// TwinCAT 3 PLC project Beispielprojekt
// ProgramVersion: 3.1.4023.0
// libraries:
//   Lynus Energy Basic, * (Lynus AG)
//   Lynus Energy ModbusTCP, * (Lynus AG)
//   Lynus Persistent Data V1, * (Lynus AG)
//   Lynus Standards, * (Lynus AG)
//   Tc2_Standard, * (Beckhoff Automation GmbH)
//   Tc2_System, * (Beckhoff Automation GmbH)
//   Tc3_Module, * (Beckhoff Automation GmbH)
//   TSG Communicator, * (EfficientIO)
// project tree:
//   / FastTask.TcTTO, PlcTask.TcTTO, SlowTask.TcTTO
//   POUs/ prgCom.TcPOU, prgCS1.TcPOU, prgEM.TcPOU, prgEMS.TcPOU (not stored), prgGrid.TcPOU, prgPD.TcPOU, prgPV.TcPOU, prgVar.TcPOU
// real-time tasks:
//   TASK FastTask: cycle T#5ms, priority 4, ADS port 350
//   TASK PlcTask: cycle T#10ms, priority 8, ADS port 351
//   TASK SlowTask: cycle T#20ms, priority 12, ADS port 352
//   TASK PlcTask1: cycle T#10ms, priority 10, ADS port 353

CONFIGURATION Beispielprojekt
    RESOURCE PLC ON TwinCAT3
        TASK FastTask(INTERVAL := T#5ms, PRIORITY := 4);
        TASK PlcTask(INTERVAL := T#10ms, PRIORITY := 8);
        TASK SlowTask(INTERVAL := T#20ms, PRIORITY := 12);
        PROGRAM prgVar WITH FastTask : prgVar;
        PROGRAM prgCS1 WITH PlcTask : prgCS1;
        PROGRAM prgEMS WITH PlcTask : prgEMS;
        PROGRAM prgGrid WITH PlcTask : prgGrid;
        PROGRAM prgPD WITH PlcTask : prgPD;
        PROGRAM prgPV WITH PlcTask : prgPV;
        PROGRAM prgEM WITH PlcTask : prgEM;
        PROGRAM prgCom WITH SlowTask : prgCom;
    END_RESOURCE
END_CONFIGURATION

// ---- POUs/prgVar.TcPOU
PROGRAM prgVar
VAR
	fbVar			: FB_VarInfo;
	fbrw1			: FB_ReadWrite;
END_VAR

fbVar(
	bReadInfo:= , 
	eTMCFile:= eSelectTMCFile.eUseTMCFile, 
	eSavePositionTMCFile:= eSavePositionOnPLC.ePostionC, 
	udiCounterFoundVariables=> , 
	bError=> , 
	bBusy=> , 
	byProgress=> , 
	udiErrorCodeOut=> , 
	eErrorVarInfo_Out=> , 
	sVarWithError=> );
	
fbrw1();

END_PROGRAM

// ---- POUs/prgCS1.TcPOU
PROGRAM prgCS1
VAR
	fbApliT_1						: FB_ECS_Alpitronic_Hypercharger;
		
	bSManualyOn_DC_1				: BOOL;												//{#lynus.ag#()}
	bEnabled_DC_1					: BOOL;												//{#lynus.ag#()}
	bySManualyTargetPowerDC_1		: BYTE;												//{#lynus.ag#()}
	bySMinPowerECSDC_1				: BYTE;												//{#lynus.ag#()}
	byErrorWarningDC_1				: BYTE;												//{#lynus.ag#()}
	lrPowerTotalDC1					: LREAL;											//{#lynus.ag#()}
	lrPowerDC1_S1					: LREAL;											//{#lynus.ag#()}
	lrPowerDC1_S2					: LREAL;											//{#lynus.ag#()}
	rChargingTimeInMinDC1_S1		: REAL;												//{#lynus.ag#()}
	rChargingTimeInMinDC1_S2		: REAL;												//{#lynus.ag#()}
	rTargetPowerDC1					: REAL;												//{#lynus.ag#()}
	dwSOCCarDC1_S1					: DWORD;											//{#lynus.ag#()}
	dwSOCCarDC1_S2					: DWORD;											//{#lynus.ag#()}
	wStateDC1_S1					: WORD;												//{#lynus.ag#()}
	wStateDC1_S2					: WORD;												//{#lynus.ag#()}
	lrEnergySessionDC1_S1			: LREAL;											//{#lynus.ag#()}
	lrEnergySessionDC1_S2			: LREAL;											//{#lynus.ag#()}
	lrTotalEnergyDC1				: LREAL;											//{#lynus.ag#()}

	fbAlfen_1						: FB_ECS_Alfen_NG9xx_Platform;
		
	bSManualyOn_Alfen_1				: BOOL;												//{#lynus.ag#()}
	bEnabled_Alfen_1				: BOOL;												//{#lynus.ag#()}
	bySManualyTargetPower_Alfen_1	: BYTE;												//{#lynus.ag#()}
	bySMinPowerECS_Alfen_1			: BYTE;												//{#lynus.ag#()}
	byErrorWarning_Alfen_1			: BYTE;												//{#lynus.ag#()}
	lrPowerTotal_Alfen_1			: LREAL;											//{#lynus.ag#()}
	lrPower_Alfen_1_S1				: LREAL;											//{#lynus.ag#()}
	lrPower_Alfen_1_S2				: LREAL;											//{#lynus.ag#()}
	rChargingTimeInMin_Alfen_1_S1	: REAL;												//{#lynus.ag#()}
	rChargingTimeInMin_Alfen_1_S2	: REAL;												//{#lynus.ag#()}
	rTargetPower_Alfen_1			: REAL;												//{#lynus.ag#()}
	wState_Alfen_1_S1				: WORD;												//{#lynus.ag#()}
	wState_Alfen_1_S2				: WORD;												//{#lynus.ag#()}
	lrEnergySession_Alfen_1_S1		: LREAL;											//{#lynus.ag#()}
	lrEnergySession_Alfen_1_S2		: LREAL;											//{#lynus.ag#()}
	lrTotalEnergy_Alfen_1			: LREAL;											//{#lynus.ag#()}
	diff_netz_pv					: LREAL;											//{#lynus.ag#()}
END_VAR
VAR PERSISTENT
	bEnableDC1						: BOOL;												//{#lynus.ag#()}
	bManualyOnDC_1					: BOOL;												//{#lynus.ag#()}
	byMinPowerDC1					: BYTE;												//{#lynus.ag#()}
	byManualyTargetPowerDC_1		: BYTE;												//{#lynus.ag#()}
	byPrioDC1						: BYTE;												//{#lynus.ag#()}
	bySOCEnableDC1					: BYTE;												//{#lynus.ag#()}
	bySOCDisableDC1					: BYTE;												//{#lynus.ag#()}
	rMaxPowerDC1					: REAL;												//{#lynus.ag#()}
	
	bEnable_Alfen_1					: BOOL;												//{#lynus.ag#()}
	bManualyOn_Alfen_1				: BOOL;												//{#lynus.ag#()}
	byMinPower_Alfen_1				: BYTE;												//{#lynus.ag#()}
	byManualyTargetPower_Alfen_1	: BYTE;												//{#lynus.ag#()}
	byPrio_Alfen_1					: BYTE;												//{#lynus.ag#()}
	bySOCEnable_Alfen_1				: BYTE;												//{#lynus.ag#()}
	bySOCDisable_Alfen_1			: BYTE;												//{#lynus.ag#()}
	rMaxPower_Alfen_1				: REAL;												//{#lynus.ag#()}
END_VAR

(*-----------------------------------------------------------------------PV vs. Netzbezug------------------------------------------------------*)
IF (lrPowerTotalDC1 + lrPowerTotal_Alfen_1) > 0 AND prgPV.lrPowerPV > (lrPowerTotalDC1 + lrPowerTotal_Alfen_1) THEN diff_netz_pv := (lrPowerTotalDC1 + lrPowerTotal_Alfen_1);
ELSIF (lrPowerTotalDC1 + lrPowerTotal_Alfen_1) > 0 AND prgPV.lrPowerPV < (lrPowerTotalDC1 + lrPowerTotal_Alfen_1) THEN diff_netz_pv := prgPV.lrPowerPV;
ELSE diff_netz_pv := 0;
END_IF

(*-----------------------------------------------------------------------Alpitronic------------------------------------------------------*)
//Manual Power
fbApliT_1.stSetupECS.bManualyOn := bManualyOnDC_1;
	fbApliT_1.stSetupECS.byManualyTargetPower := byManualyTargetPowerDC_1;
		fbApliT_1.stSetupECS.byPriority := byPrioDC1;
			fbApliT_1.stSetupECS.byEnableSOC := bySOCEnableDC1;
				fbApliT_1.stSetupECS.byDisableSOC := bySOCDisableDC1;
					fbApliT_1.stSetupECS.rMaxPower := rMaxPowerDC1;
						fbApliT_1.stSetupECS.byCSMinPower := byMinPowerDC1;	
	
fbApliT_1(
	bEnable:= bEnableDC1, 
	bPowerDataInvers:= , 
	byElectricFuseLine:= , 
	byUnitID:= 1, 	//Normaly always 1 for Alpitronic
	diNrOfEMS_IN:= prgEMS.fbEMS.diNrOfEMS_OUT, 
	diNrOfEM_IN_CS:= , 
	sIPAdress:= '172.16.1.110', 
	stSetupECS:= , 
	stDataECS=> , 
	diNrOfECS_OUT=> );

bSManualyOn_DC_1 := fbApliT_1.stDataECS.bSManualyOn;
	bySManualyTargetPowerDC_1 := fbApliT_1.stDataECS.bySManualyTargetPower;
		byErrorWarningDC_1 := fbApliT_1.stDataECS.byErrorWarning;
			lrPowerTotalDC1 := fbApliT_1.stDataECS.lrTotalPower;
				lrPowerDC1_S1 :=  fbApliT_1.stDataECS.arrSocketPower[1];
					lrPowerDC1_S2 :=  fbApliT_1.stDataECS.arrSocketPower[2];	 	
						rChargingTimeInMinDC1_S1 := fbApliT_1.stDataECS.arrChargingTimeInMin[1];	
							rChargingTimeInMinDC1_S2 := fbApliT_1.stDataECS.arrChargingTimeInMin[2];
								dwSOCCarDC1_S1 := fbApliT_1.stDataECS.arrSocketSOCCar[1]; 
									dwSOCCarDC1_S2 := fbApliT_1.stDataECS.arrSocketSOCCar[2]; 	
										wStateDC1_S1 := fbApliT_1.stDataECS.arrSocketStateECS[1];
											wStateDC1_S2 := fbApliT_1.stDataECS.arrSocketStateECS[2];
												lrEnergySessionDC1_S1 := fbApliT_1.stDataECS.arrSocketEnergySession[1];
													lrEnergySessionDC1_S2 := fbApliT_1.stDataECS.arrSocketEnergySession[2];
														lrTotalEnergyDC1 := fbApliT_1.stDataECS.lrTotalCounterEnergy_Consumption;
															bySMinPowerECSDC_1 := fbApliT_1.stDataECS.bySCSMinPower;
																rTargetPowerDC1 := fbApliT_1.stDataECS.rTargetPower;
																	bEnabled_DC_1 := fbApliT_1.stDataECS.bEnabled;
																	
(*-----------------------------------------------------------------------Alfen------------------------------------------------------*)

//Manual Power
fbAlfen_1.stSetupECS.bManualyOn := bManualyOn_Alfen_1;
	fbAlfen_1.stSetupECS.byManualyTargetPower := byManualyTargetPower_Alfen_1;
		fbAlfen_1.stSetupECS.byPriority := byPrio_Alfen_1;
			fbAlfen_1.stSetupECS.byEnableSOC := bySOCEnable_Alfen_1;
				fbAlfen_1.stSetupECS.byDisableSOC := bySOCDisable_Alfen_1;
					fbAlfen_1.stSetupECS.rMaxPower := rMaxPower_Alfen_1;
						fbAlfen_1.stSetupECS.byCSMinPower := byMinPower_Alfen_1;	
	
fbAlfen_1(
	bEnable:= bEnable_Alfen_1, 
	bPowerDataInvers:= , 
	byElectricFuseLine:= , 
	byUnitID_Socket1:= 1, 
	byUnitID_Socket2:= 2, 
	byNumberOfSockets:= 2,		//1 or 2. Depends on whether it is a single or double charging station  
	byNumberOfConnectionWire:= 2, //1 or 2.  Depends on whether the charging station is supplied via a supply line or
	diNrOfEMS_IN:= prgEMS.fbEMS.diNrOfEMS_OUT, 
	diNrOfEM_IN_CS:= , 
	sIPAdress:= '172.16.1.100', 
	stSetupECS:= , 
	stDataECS=> , 
	diNrOfECS_OUT=> , 
	lrTotalPowerECSRealTime=> );						
						
bSManualyOn_Alfen_1 := fbAlfen_1.stDataECS.bSManualyOn;
	bySManualyTargetPower_Alfen_1 := fbAlfen_1.stDataECS.bySManualyTargetPower;
		byErrorWarning_Alfen_1 := fbAlfen_1.stDataECS.byErrorWarning;
			lrPowerTotal_Alfen_1 := fbAlfen_1.stDataECS.lrTotalPower;
				lrPower_Alfen_1_S1 :=  fbAlfen_1.stDataECS.arrSocketPower[1];
				lrPower_Alfen_1_S2 :=  fbAlfen_1.stDataECS.arrSocketPower[2];
					rChargingTimeInMin_Alfen_1_S1 := fbAlfen_1.stDataECS.arrChargingTimeInMin[1];
					rChargingTimeInMin_Alfen_1_S2 := fbAlfen_1.stDataECS.arrChargingTimeInMin[2];	
						wState_Alfen_1_S1 := fbAlfen_1.stDataECS.arrSocketStateECS[1];
						wState_Alfen_1_S2 := fbAlfen_1.stDataECS.arrSocketStateECS[2];
							lrEnergySession_Alfen_1_S1 := fbAlfen_1.stDataECS.arrSocketEnergySession[1];
							lrEnergySession_Alfen_1_S1 := fbAlfen_1.stDataECS.arrSocketEnergySession[2];
								lrTotalEnergy_Alfen_1 := fbAlfen_1.stDataECS.lrTotalCounterEnergy_Consumption;
									bySMinPowerECS_Alfen_1 := fbAlfen_1.stDataECS.bySCSMinPower;
										rTargetPower_Alfen_1 := fbAlfen_1.stDataECS.rTargetPower;
											bEnabled_Alfen_1 := fbAlfen_1.stDataECS.bEnabled;

END_PROGRAM

// ---- POUs/prgPV.TcPOU
PROGRAM prgPV
VAR
	fbPV1					: FB_Firmer_PV_Inverter_Sunspec;
	fbPV2					: FB_Firmer_PV_Inverter_Sunspec;
	fbPVInt1				: FB_PV_Power;
	fbPVInt2				: FB_PV_Power;
	fbPVCounter				: FB_EnergyCounter;
	lrPowerPV				: LREAL;				//{#lynus.ag#()}
	lrPowerPV1				: LREAL;				//{#lynus.ag#()}
	lrPowerPV2				: LREAL;				//{#lynus.ag#()}
	byErrorWarningPV1		: BYTE;					//{#lynus.ag#()}
	byErrorWarningPV2		: BYTE;					//{#lynus.ag#()}
END_VAR
VAR PERSISTENT
	lrCounterPV				: LREAL;				//{#lynus.ag#()}
END_VAR

fbPV1(
	bEnable:= TRUE, 
	sIPAdress:= '172.16.1.161',
	byUnitID_Inverter := 1,
	stFirmerInverterData=> , 
	stDataEMPower_PV=> , 
	stDataEMCounter_PV=> , 
	diNrOfEM_OUT_PV=> );

fbPV2(
	bEnable:= TRUE, 
	sIPAdress:= '172.16.1.162',
	byUnitID_Inverter := 1,
	stFirmerInverterData=> , 
	stDataEMPower_PV=> , 
	stDataEMCounter_PV=> , 
	diNrOfEM_OUT_PV=> );
	
fbPVInt1(
	bEnable:= TRUE, 
	bPowerDataInvers:= , 
	diNrOfEM_IN_PV:= fbPV1.diNrOfEM_OUT_PV, 
	stDataPv=> , 
	diNrOfPv_OUT=> );

fbPVInt2(
	bEnable:= TRUE, 
	bPowerDataInvers:= , 
	diNrOfEM_IN_PV:= fbPV2.diNrOfEM_OUT_PV, 
	stDataPv=> , 
	diNrOfPv_OUT=> );

lrPowerPV1 := fbPVInt1.stDataPv.lrPower;
lrPowerPV2 := fbPVInt2.stDataPv.lrPower;
	byErrorWarningPV1 := fbPVInt1.stDataPv.byErrorWarning;
	byErrorWarningPV2 := fbPVInt2.stDataPv.byErrorWarning;

// PV Power Total
lrPowerPV := fbPVInt1.stDataPv.lrPower + fbPVInt2.stDataPv.lrPower;


// EnergyCounter (Total)
fbPVCounter(
	byActiveTariff:= 1, 
	lrPowerInput:= 0 - lrPowerPV, 
	lrTotalCounterEnergy_Consumption=> , 
	lrTotalCounterEnergy_Production=> , 
	lrCounterEnergyT1_Consumption=> , 
	lrCounterEnergyT2_Consumption=> , 
	lrCounterEnergyT1_Production=> , 
	lrCounterEnergyT2_Production=> );
	
IF fbPVCounter.lrTotalCounterEnergy_Production > lrCounterPV THEN  	
	lrCounterPV := fbPVCounter.lrTotalCounterEnergy_Production;
END_IF

END_PROGRAM

// ---- POUs/prgGrid.TcPOU
PROGRAM prgGrid
VAR PERSISTENT
	rSizeGridConn				: REAL;									//{#lynus.ag#()}
END_VAR
VAR
	fbGrid						: FB_Grid_Power_Ext_Input;
	lrGridPower					: LREAL;								//{#lynus.ag#()}
END_VAR

IF prgEM.fbEM.stDataEMPowerRealTime.byErrorWarning = 2 THEN fbGrid.bExtErrorGrid := TRUE; ELSE fbGrid.bExtErrorGrid := FALSE; END_IF

fbGrid(
	bEnable:= TRUE, 
	diNrOfEMS_IN:= prgEMS.fbEMS.diNrOfEMS_OUT, 
	rSizeGridConn:= rSizeGridConn, 
	bExtErrorGrid:= , 
	lrExtGridPower:= prgEM.fbEM.stDataEMPowerRealTime.lrPowerTotal, 
	lrExtTotalCounterEnergy_Consumption:= 0, 
	lrExtTotalCounterEnergy_Production:= 0, 
	lrExtCounterEnergyT1_Consumption:= 0, 
	lrExtCounterEnergyT2_Consumption:= 0, 
	lrExtCounterEnergyT1_Production:= 0, 
	lrExtCounterEnergyT2_Production:= 0,
	stDataGrid=> ,
	diNrOfGrid_OUT=> );
	
lrGridPower := fbGrid.stDataGrid.lrPower;

END_PROGRAM

// ---- POUs/prgEM.TcPOU
PROGRAM prgEM
VAR
	fbEM				: FB_PhoenixContact_EM_EEM_EM375;
	lrEMPowerTotal		: LREAL;
END_VAR
VAR PERSISTENT
	bEnableEM			: BOOL;
	lrEMCounterProd		: LREAL;
	lrEMCounterCons		: LREAL;
END_VAR

fbEM(
	bEnable:=bEnableEM,
	byUnitID:=255,
	sIPAdress:='172.16.1.151',
	diNrOfEM_OUT=>,
	stDataEMPowerRealTime=>,
	stDataEMCounterRealTime=>);

lrEMPowerTotal := fbEM.stDataEMPowerRealTime.lrPowerTotal;
	lrEMCounterProd := fbEM.stDataEMCounterRealTime.lrTotalCounterEnergy_Production;
		lrEMCounterCons := fbEM.stDataEMCounterRealTime.lrTotalCounterEnergy_Consumption;

END_PROGRAM

// ---- POUs/prgPD.TcPOU
PROGRAM prgPD
VAR
	fbPers						: FB_WritePersistentData_General;
END_VAR

fbPers(
	eSaveModeData:= eUSVSaveMode.eSaveEventBased, 
	bLoadPersistentDataOk=> , 
	bError=> , 
	bySaveProcess=> , 
	dwStorageLast24h=> , 
	udiErrorCode=> );

END_PROGRAM

// ---- POUs/prgCom.TcPOU
PROGRAM prgCom
VAR
	fbCom			: FB_MqttCommunicator;
END_VAR

fbCom(
	bConnect:= TRUE, 
	sUserName:= 'dd42716e-193d-4c6c-a2c4-46c477e1877b', 
	sUserPassword:= 'b13d7ac3-0642-4711-8449-ebfd8a27b319', 
	eSavePositionCertificate:= eSavePositionOnPLC.ePostionC, 
	bConnected=> , 
	bError=> , 
	hrErrorCode=> , 
	eConnectionState=> , 
	eErrorMessage_Out=> );

END_PROGRAM
